// TIA Portal V17 export
// export: Created 2026-05-13T14:55:42.2439207Z, ExportSetting WithDefaults, DisplayName Totally Integrated Automation Portal, DisplayVersion V17 Update 4, DisplayName TIA Portal Openness, DisplayVersion V17 Update 4, DisplayName TIA Portal Version Control Interface, DisplayVersion V17, DisplayName SINAMICS Startdrive Advanced, DisplayVersion V17, DisplayName SINAMICS Startdrive G130, G150, S120, S150, SINAMICS MV, S210, DisplayVersion V17, DisplayName SINAMICS Startdrive G110M, G120, G120C, G120D, G120P, G115D, DisplayVersion V17, DisplayName STEP 7 Professional, DisplayVersion V17 Update 4, DisplayName STEP 7 Safety, DisplayVersion V17, DisplayName WinCC Professional, DisplayVersion V17 Update 4
DATA_BLOCK "DB_Components"   // DB2
{ S7_Optimized_Access := 'TRUE' }
VERSION : 0.1
// stored: AutoNumber true, DBAccessibleFromOPCUA true, DBAccessibleFromWebserver true, IsOnlyStoredInLoadMemory false, IsRetainMemResEnabled false, IsWriteProtectedInAS false, MemoryReserve 100
   VAR
      Valve01 { S7_SetPoint := 'True'} : "UDT_ComponentPopup";   // 阀门
      Heater01 { S7_SetPoint := 'True'} : "UDT_ComponentPopup";   // 电加热
      Fan01 { S7_SetPoint := 'True'} : "UDT_ComponentPopup";   // 循环风机
   END_VAR
BEGIN
   Valve01.InfoTitle := '阀门01';
   Valve01.InfoMessage := '是否确认开启阀门01？';
   Heater01.InfoTitle := '电加热01';
   Heater01.InfoMessage := '是否确认开启电加热01？';
   Fan01.InfoTitle := '循环风机01';
   Fan01.InfoMessage := '是否确认开启循环风机01？';
END_DATA_BLOCK
